Staubli VAL3: setItem.pgx

public program setItem(InstrItem& x_sItem[], num& x_nIndex[])
begin
  // set IT
  pEdit.iEvent[x_nIndex]=x_sItem
end
